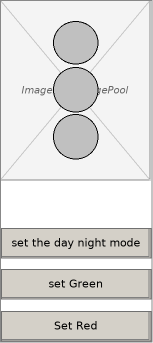
VISUALIZATION TrafficLightVPrototype  // 153x343
VAR_IN_OUT
	stTrafficIn : ST_TrafficLightInput;
	stTrafficOut : ST_TrafficLightOutput;
END_VAR
    Image (0,0 150x180), image: ImagePool.ImagePool
    Ellipse (53,67 45x45), colour toggle: stTrafficOut.bYellow
    Ellipse (53,21 45x43), colour toggle: stTrafficOut.bRed
    Ellipse (53,114 45x45), colour toggle: stTrafficOut.bGreen
    Button (1,228 150x30), "set the day night mode"
        toggle MAIN.fbCrossing1.bCDayMode
    Button (1,269 150x30), "set Green"
        tap stTrafficIn.bSetGreen
    Button (1,311 150x30), "Set Red"
        tap stTrafficIn.bSetRed
END_VISUALIZATION

(* stored: Version 1.1.0.1, ProductVersion 3.1.4024.0
   Visu TrafficLightVPrototype: Id {c86a29df-a886-4e95-9763-ab21492b4201} *)
